// writes traces into files, deletes too old files and monitors hdd usage
{attribute 'reflection'}
FUNCTION_BLOCK PUBLIC FB_TraceHandler IMPLEMENTS I_TraceHandler
(**************************************************************************************
 *  Application     : BoxControl Framework
 *  Revision        : $Revision: 404529 $
 *  Revision date   : $Date: 2020-10-20 08:21:38 +0200 (Mo., 20 Oct 2020) $
 *  Last changed by : $Author: b7lipim $
 *  URL             : $URL: http://almscdc.swisslog.com/repo/SWPD/Development/BoxControlFramework/20_Release/trunk/01_Software/BCF/BCF/JumpStart/20_Product/10_App/11_Com/10_Lib/FB_DebugMsg.TcPOU $
 *
 *  Purpose :	writes (debug) messages into files in subfolders
 *            deletes all subfolders including files older than 7d (according to name, not date)
 *            monitors hdd usage, reports it via debug message and surpress further writing if 80% is exceeded
 *
 * ------------------------------------------------------------------------------------
 *  Copyright Swisslog [IP AG], Switzerland. All rights reserved.
 * 
 * ------------------------------------------------------------------------------------
 *	
 * 	Revision History: 
 *
 *  VERSION DATE         INITIALS     DESCRIPTION
 *  0.0     DD.MM.YYYY   (name)       (explain customized modifications)
 *
 **************************************************************************************)

(********************************************************************************************************************************)
VAR_STAT CONSTANT
  SHELF_LIFE            : TIME                             := T#7D;      // duration until old folders will be deleted
  (*----------------------------------------------------------------------------------------------------------------------------*)
  MAX_FILEOPEN_TIME     : TIME                             := T#100MS;   // maximum file open time until reopen/flush
  LOCKTIME              : TIME                             := T#100MS;   // inhibit time between write attemts
  (*----------------------------------------------------------------------------------------------------------------------------*)
  BUFFER_SIZE           : WORD                             := 8192;      // size of internal file write buffer
  FIFO_SIZE             : WORD                             := 1024;      // size of internal dynamic fifo to temporary store trace entries
  (*----------------------------------------------------------------------------------------------------------------------------*)
  HDD_WARNING_LEVEL     : BYTE                             := 60;        // warning if hdd usage exceeds this percentage
  HDD_ERROR_LEVEL       : BYTE                             := 80;        // error and stop writing if hdd usage exceeds this percentage
END_VAR

(********************************************************************************************************************************)
VAR
  {attribute 'instance-path'}
  {attribute 'no_init'}
  _Instance             : STRING[255]                      := '';         // instance path
  (*----------------------------------------------------------------------------------------------------------------------------*)
  _Enable               : BOOL                             := FALSE;      // HI = writing/deleting enabled
  _MaxFileSizeKB        : WORD                             := 10_240;     // maximum file size in kilobytes
  _Folder               : A_TracePath                      := '';         // working folder without ending '/'
  (*-- duration ----------------------------------------------------------------------------------------------------------------*)
  _StartSystemTick      : ULINT                            := 0;          // system tick at execution start
  _GetSystemTicks       : GETCPUCOUNTER;                                  // Gets the system time in 100ns ticks  
  (*-- general -----------------------------------------------------------------------------------------------------------------*)
  _GetHostName          : FB_GetHostName()                 := (sNetID:= '', tTimeout:= DEFAULT_ADS_TIMEOUT);
  _GetAdaptersInfo      : FB_GetAdaptersInfo()             := (sNetID:= '', tTimeout:= DEFAULT_ADS_TIMEOUT);
  _GetDeviceIdentificationEx : FB_GetDeviceIdentificationEx:= (sNetID:= '', tTimeout:= DEFAULT_ADS_TIMEOUT);
  _MainFolder           : A_TracePath                      := '';         // working folder ending without '/'
  _Active               : BOOL                             := FALSE;      // HI = enable and working folder exists
  _Opened               : BOOL                             := FALSE;      // HI = file is currently open
  _PlcRestarted         : BOOL                             := TRUE;       // HI = add separation lines to file
  _MillisecondsLast		: WORD                             := 16#FFFF;    // system clock monitoring
  _Text                 : STRING[255]                      := '';         // own debug message
  (*-- checking work folder - states -------------------------------------------------------------------------------------------*)
  _CheckState           : E_TraceCheckStates               := E_TraceCheckStates.Initialization;
  _CheckStateLast       : E_TraceCheckStates               := E_TraceCheckStates.Initialization;
  _CheckTime            : TIME                             := T#0S;
  (*-- writing files - states --------------------------------------------------------------------------------------------------*)
  _WriteState           : E_TraceWriteStates               := E_TraceWriteStates.Initialization;
  _WriteStateLast       : E_TraceWriteStates               := E_TraceWriteStates.Initialization;
  _WriteTime            : TIME                             := T#0S;
  (*-- deleting files - states -------------------------------------------------------------------------------------------------*)
  _DeleteState          : E_TraceDeleteStates              := E_TraceDeleteStates.Initialization;
  _DeleteStateLast      : E_TraceDeleteStates              := E_TraceDeleteStates.Initialization;
  _DeleteTime           : TIME                             := T#0S;
  (*-- hdd monitoring ----------------------------------------------------------------------------------------------------------*)
  _HddUsage             : FB_HddUsage;
  _HddUsageTime         : TIME                             := T#0S;
  _HddUsageCount        : DWORD                            := 0;               // counter
  _HddState             : E_TraceHddUsageStates            := E_TraceHddUsageStates.Initialization;
  _HddStateLast         : E_TraceHddUsageStates            := E_TraceHddUsageStates.Initialization;
  _HddTooFull           : BOOL                             := FALSE;           // hdd is too full to write
  _HddFullMissed        : ULINT                            := 0;               // rejected messages due to hdd too full  ( maybe persistent? )
  (*-- writing files - data ----------------------------------------------------------------------------------------------------*)
  _WritePath            : A_TracePath                      := '';              // current working folder with date and trailing '/'
  _WriteFileName        : A_TracePath                      := '';              // current file name
  _WriteDate            : TIMESTRUCT;                                          // current working date
  (*-- file handling -----------------------------------------------------------------------------------------------------------*)
  _FileSize             : ULINT                            := 0;               // current file size in bytes
  _FileIndex            : WORD                             := 0;               // current file number
  _FileTimeOpened       : TIME                             := T#0S;            // timestamp file was opened
  _CreateDir            : Tc2_System.FB_CreateDir;                             // create new folder
  _FileCheck            : Tc2_Utilities.FB_EnumFindFileEntry;                  // checks current working folder for already existing files
  _FileOpen             : Tc2_System.FB_FileOpen;                              // open/create file
  _FileWrite            : Tc2_System.FB_FileWrite;                             // write into file
  _FileClose            : Tc2_System.FB_FileClose;                             // close file
  (*-- folder handling ---------------------------------------------------------------------------------------------------------*)
  _CheckWorkFolder      : Tc2_Utilities.FB_EnumFindFileEntry;                  // checks working folder being existent
  _ScanSubFolder        : Tc2_Utilities.FB_EnumFindFileEntry;                  // checks current working folder for subfolders
  _FileFind             : Tc2_Utilities.FB_EnumFindFileEntry;                  // checks (old) subfolders for files to delete
  _FileDelete           : Tc2_System.FB_FileDelete;                            // delete file
  _FolderRemove         : Tc2_System.FB_RemoveDir;                             // delete folder
  (*-- write fifo --------------------------------------------------------------------------------------------------------------*)
  _TaskCounter          : WORD                             := 0;               // counter for put calls within one plc cycle
  _FifoFillLevel        : WORD                             := 0;               // fill level
  _FifoInput            : WORD                             := 0;               // (next) input position
  _FifoOutput           : WORD                             := 0;               // (next) output position
  _Fifo                 : ARRAY[0..FIFO_SIZE-1] OF POINTER TO FB_TraceEntry;          // fifo itself
  (*-- write data --------------------------------------------------------------------------------------------------------------*)
  _DataDateChanged      : BOOL                             := FALSE;           // date of write data has changed
  _DataLength           : DWORD                            := 0;               // valid length of _DataBuffer
  _DataBuffer           : ARRAY[0..BUFFER_SIZE-1] OF BYTE;                     // data buffer to write into file
  (*-- diagnostics & statisticals ------------------------------------------------------------------------------------------------*)
  _Statistics           : FB_TraceHandlerStatistics();
  _ExecutionDuration    : ULINT                            := 0;               // duration of execution in microseconds
  _ExecutionNow         : ULINT                            := 0;
  (*-- testing -------------------------------------------------------------------------------------------------------------------*)
  _Diag_SystemTime      : ULINT                            := 0;
  _Diag_NoMemory        : ULINT                            := 0;
  _Diag_NoEntry         : ULINT                            := 0;
  _Diag_FifoFull        : ULINT                            := 0;
  _Diag_InvalidDate     : ULINT                            := 0;
END_VAR

(*****************************************************1*********2*********3*********4*********5*********6*********7*********8****)
VAR_STAT CONSTANT                          // 123456789012345678901234567890123456789012345678901234567890123456789012345678900123456789001234567890
{attribute 'hide'}  EOF      : STRING[ 95]:= ';-- end of file ----------------------------------------------------------------';
{attribute 'hide'}  NEWLINE  : STRING[  3]:= '$0D$0A';
{attribute 'hide'}  DIVIDER  : STRING[ 95]:= ';-------------------------------------------------------------------------------';
{attribute 'hide'}  CREATED  : STRING[ 15]:= '; CREATED  : ';
{attribute 'hide'}  TD       : STRING[ 15]:= '; DATE     : ';
{attribute 'hide'}  ENCODING : STRING[ 19]:= '; ENCODING : UTF08';
{attribute 'hide'}  EMPTYLINE: STRING[  3]:= '; ';
{attribute 'hide'}  APPL     : STRING[ 15]:= '; APPL     : ';
{attribute 'hide'}  BUILD    : STRING[ 15]:= '; BUILD    : ';
{attribute 'hide'}  HOST     : STRING[ 15]:= '; HOST     : ';
{attribute 'hide'}  ADDR     : STRING[ 15]:= '; ADDR     : ';
{attribute 'hide'}  OPSYSTEM : STRING[ 15]:= '; SYSTEM   : ';
{attribute 'hide'}  RUNTIME  : STRING[ 19]:= '; RUNTIME  : TC';
{attribute 'hide'}  INFO     : STRING[ 15]:= '; INFO     : ';
{attribute 'hide'}  SIZE     : STRING[ 15]:= '; SIZE     : ';
{attribute 'hide'}  HEADER   : STRING[195]:= '; -- DATE & TIME ------- count -- level -- instance -------------------------- position ------- message ------- additional information ------';
END_VAR


(********************************************************************************************************************************)
(** calculate execution time ****************************************************************************************************)
_GetSystemTicks();
_StartSystemTick:= (         DWORD_TO_ULINT(_GetSystemTicks.cpuCntLoDW)
                     OR SHL( DWORD_TO_ULINT(_GetSystemTicks.cpuCntHiDW),  32 )  );




(********************************************************************************************************************************)
(** run all services ************************************************************************************************************)
_HddUsage();  // call here to use everywhere

M_RunHddUsage();
M_RunCheck();
M_RunWrite();
M_RunDelete();

IF (_MillisecondsLast = System.fbSystemTime.TIMESTR.wMilliseconds)
THEN
  _Diag_SystemTime:= _Diag_SystemTime + 1;

  (*-- trace it ---------------------------------------------------*)
  IF(_TaskCounter <> 0)
  THEN
// example: '11-000-0000-00-0,  system time not updated'
   ;(* _Text:= '';
    _Text:= CONCAT(_Text, F_AddDividerToSisString(SubsystemRegistry.SubsystemName) );
    _Text:= CONCAT(_Text, ',  system time not updated');
    Put( MsgType := E_DebugMsgType.WARNING,
         Instance:= ADR(_Instance),
         Text    := ADR(_Text)  );*)
  END_IF
END_IF

_MillisecondsLast:= System.fbSystemTime.TIMESTR.wMilliseconds;
_TaskCounter:= 0;




(********************************************************************************************************************************)
(** calculate execution time ****************************************************************************************************)
_GetSystemTicks();

_ExecutionNow:= (         DWORD_TO_ULINT(_GetSystemTicks.cpuCntLoDW)
                  OR SHL( DWORD_TO_ULINT(_GetSystemTicks.cpuCntHiDW),  32 )  );

_ExecutionDuration:= (_ExecutionNow - _StartSystemTick + 5) / 10;

_Statistics.MaxExecutionDuration:= MAX(_Statistics.MaxExecutionDuration, _ExecutionDuration);




(********************************************************************************************************************************)
(** done ************************************************************************************************************************)

// clears the internal fifo (all unwritten traces will be lost)
METHOD PUBLIC Clear

(********************************************************************************************************************************)
VAR_INPUT
END_VAR

(********************************************************************************************************************************)
VAR
  Index                 : WORD                             := 0;
  Entry                 : POINTER TO FB_TraceEntry         := 0;
END_VAR

(********************************************************************************************************************************)
(********************************************************************************************************************************)
_FifoFillLevel:= 0;
_FifoInput    := 0;
_FifoOutput   := 0;




(********************************************************************************************************************************)
(********************************************************************************************************************************)
Index:= 0;
WHILE (Index < FIFO_SIZE)
DO
  Entry:= _Fifo[Index];

  (*-- release memory -----------------------------------------------*)
  IF (Entry <> 0)
  THEN
    __DELETE(Entry);
  END_IF

  (*-- next ---------------------------------------------------------*)
  _Fifo[Index]:= 0;
  Index:= Index + 1;
END_WHILE




(********************************************************************************************************************************)
(** done ************************************************************************************************************************)
END_METHOD

// HI = writing/deleting enabled
{attribute 'monitoring' := 'call'}
PROPERTY PUBLIC Enable : BOOL
GET
Enable:= _Enable;
END_GET
SET
(********************************************************************************************************************************)
(** change? *********************************************************************************************************************)
IF (_Enable = Enable)
THEN
  RETURN;
END_IF

_Enable:= Enable;




(********************************************************************************************************************************)
(** done ************************************************************************************************************************)
END_SET
END_PROPERTY

{attribute 'hide'}
METHOD FB_exit : BOOL

(********************************************************************************************************************************)
VAR_INPUT
	bInCopyCode           : BOOL;  // if TRUE, the instance afterwards gets moved into the copy code (online change)
  (*----------------------------------------------------------------------------------------------------------------------------*)
END_VAR

(********************************************************************************************************************************)
(** release dynamically assigned memory *****************************************************************************************)
Clear();




(********************************************************************************************************************************)
(** done ************************************************************************************************************************)
END_METHOD

{attribute 'hide'}
METHOD FB_init : BOOL

(********************************************************************************************************************************)
VAR_INPUT
	bInitRetains          : BOOL; // if TRUE, the retain variables are initialized (warm start / cold start)
	bInCopyCode           : BOOL;  // if TRUE, the instance afterwards gets moved into the copy code (online change)
  (*----------------------------------------------------------------------------------------------------------------------------*)
END_VAR

(********************************************************************************************************************************)
VAR
END_VAR

(********************************************************************************************************************************)
(** remove 'QB2Jumpstart.JumpStart.' from instance path *************************************************************************)
F_InstancePathRemovals( DestStart     := ADR(_Instance),
                        DestEnd       := ADR(_Instance) + SIZEOF(_Instance),
                        RemoveLastPart:= FALSE );




(********************************************************************************************************************************)
(** done ************************************************************************************************************************)
END_METHOD

// folder to work within, folder must exist! (will only take effect when enabled is low)
{attribute 'monitoring' := 'call'}
PROPERTY PUBLIC Folder : A_TracePath
GET
Folder:= _Folder;
END_GET
SET
VAR
  Idx                   : WORD                             := 0;
  SepFound              : BOOL                             := FALSE;
  Finished              : BOOL                             := FALSE;
END_VAR
(********************************************************************************************************************************)
(** change? *********************************************************************************************************************)
IF (_Folder = Folder)
THEN
  RETURN;
END_IF

_Folder:= Folder;




(********************************************************************************************************************************)
(** change '\' to '/' and remove a trailing '/' if neccessary *******************************************************************)
Idx:= 0;
WHILE (Idx < SIZEOF(_Folder)  )
DO
  (*-- replace '\' with '/' -------------------------------------------------------------*)
  IF (_Folder[Idx] = 16#5C)  (* '\' *)
  THEN
    _Folder[Idx]:= 16#2F;   (* '/' *)
    SepFound:= TRUE;

  (*-- separation found '/' -------------------------------------------------------------*)
  ELSIF(_Folder[Idx] = 16#2F)   (* '/' *)
  THEN
    SepFound:= TRUE;

  (*-- fill rest of string with terminations --------------------------------------------*)
  ELSIF(Finished = TRUE)
  THEN
    (*-------------------------------------------*)
    _Folder[Idx]:= 16#00;

  (*-- string termination found ---------------------------------------------------------*)
  ELSIF(_Folder[Idx] = 16#00)
  THEN
    (*-- remove trailing '/' --------------------*)
    IF (SepFound = TRUE)
    THEN
      _Folder[Idx-1] := 16#00;
    END_IF
    (*-------------------------------------------*)
    Finished:= TRUE;
    SepFound:= FALSE;

  (*-- normal character -----------------------------------------------------------------*)
  ELSE
    SepFound:= FALSE;
  END_IF

  (*-- next -----------------------------------------------------------------------------*)
  Idx:= Idx + 1;
END_WHILE




(********************************************************************************************************************************)
(** done ************************************************************************************************************************)
END_SET
END_PROPERTY

// usage/free and total space of hdd
{attribute 'monitoring' := 'call'}
PROPERTY PUBLIC HddUsage : I_HddUsage
GET
HddUsage:= _HddUsage;
END_GET
END_PROPERTY

// builds the file name with index
METHOD PROTECTED M_BuildFileName

(********************************************************************************************************************************)
VAR
  DestStart             : POINTER TO BYTE                  := 0;     // start position to concat
  DestEnd               : POINTER TO BYTE                  := 0;     // buffer/string end
END_VAR

(********************************************************************************************************************************)
(********************************************************************************************************************************)
DestStart:= ADR(_WriteFileName);
DestEnd  := ADR(_WriteFileName) + SIZEOF(_WriteFileName);

(*-- application ---------------------------------------------------------------------------------------------------------------*)
DestStart:= F_StringCopy          ( DestStart:= DestStart,  DestEnd:= DestEnd,  Source    := ADR(_GetHostName.sHostName)  );

(*-- date ----------------------------------------------------------------------------------------------------------------------*)
DestStart:= F_StringCopy          ( DestStart:= DestStart,  DestEnd:= DestEnd,  Source    := ADR('_')  );
DestStart:= F_StringFromDatestruct( DestStart:= DestStart,  DestEnd:= DestEnd,  DateStruct:= _WriteDate );

(*-- index ---------------------------------------------------------------------------------------------------------------------*)
DestStart:= F_StringCopy          ( DestStart:= DestStart,  DestEnd:= DestEnd,  Source    := ADR('_')  );
DestStart:= F_StringFromWord      ( DestStart:= DestStart,  DestEnd:= DestEnd,  Value     := _FileIndex,  Length:= 4 );


(*-- file type -----------------------------------------------------------------------------------------------------------------*)
DestStart:= F_StringCopy          ( DestStart:= DestStart,  DestEnd:= DestEnd,  Source    := ADR('_Trace.txt')  );




(********************************************************************************************************************************)
(** done ************************************************************************************************************************)
END_METHOD

// created data to write, returns TRUE if trace date has changed
METHOD PROTECTED M_CreateData : BOOL

(********************************************************************************************************************************)
VAR
  MsgText               : STRING[31]                       := ''; 
  (*----------------------------------------------------------------------------------------------------------------------------*)
  DestStart             : POINTER TO BYTE                  := 0;
  DestWork              : POINTER TO BYTE                  := 0;
  DestEnd               : POINTER TO BYTE                  := 0;
  (*----------------------------------------------------------------------------------------------------------------------------*)
  EntryStart            : POINTER TO BYTE                  := 0;
  Entry                 : POINTER TO FB_TraceEntry         := 0;
  DateChanged           : BOOL                             := FALSE;
  Count                 : WORD                             := 0;
END_VAR

(********************************************************************************************************************************)
(********************************************************************************************************************************)
_DataLength:= 0;

DestStart:= ADR(_DataBuffer);
DestWork := ADR(_DataBuffer);
DestEnd  := ADR(_DataBuffer) + SIZEOF(_DataBuffer);

DateChanged:= FALSE;




(********************************************************************************************************************************)
(********************************************************************************************************************************)
Count:= 0;
WHILE(_FifoFillLevel <> 0)
DO
  (*-- get new entry --------------------------------------------------------------------*)
  Entry:= _Fifo[_FifoOutput];
  IF (Entry = 0)
  THEN
    EXIT;
  END_IF

  (*-- entry has already new date? ------------------------------------------------------*)
  IF (Entry^.IsEqualDate(_WriteDate) = FALSE)
  THEN
    DateChanged:= TRUE;
    EXIT;
  END_IF

  (*-- prepare line ---------------------------------------------------------------------*)
  MsgText:= TO_STRING(Entry^.MsgType);

  (*-- build line -----------------------------------------------------------------------*)
  EntryStart:= DestWork;
  DestWork:= F_StringFromDatestruct( DestStart:= DestWork,  DestEnd:= DestEnd,  DateStruct:= Entry^.DateTime  );
  DestWork:= F_StringCopy          ( DestStart:= DestWork,  DestEnd:= DestEnd,  Source    := ADR('  ')  );
  DestWork:= F_StringFromTimestruct( DestStart:= DestWork,  DestEnd:= DestEnd,  TimeStruct:= Entry^.DateTime,     ShowMs:= TRUE  );
  DestWork:= F_StringCopy          ( DestStart:= DestWork,  DestEnd:= DestEnd,  Source    := ADR(':  ')  );
  DestWork:= F_StringFromWord      ( DestStart:= DestWork,  DestEnd:= DestEnd,  Value     := Entry^.TaskCounter,  Length:= 0  );
  DestWork:= F_StringCopy          ( DestStart:= DestWork,  DestEnd:= DestEnd,  Source    := ADR(' = ')  );
  DestWork:= F_StringCopy          ( DestStart:= DestWork,  DestEnd:= DestEnd,  Source    := ADR(MsgText)  );
  DestWork:= F_StringCopy          ( DestStart:= DestWork,  DestEnd:= DestEnd,  Source    := ADR(',  ')  );
  DestWork:= F_StringCopy          ( DestStart:= DestWork,  DestEnd:= DestEnd,  Source    := Entry^.InstancePtr); 
  DestWork:= F_StringCopy          ( DestStart:= DestWork,  DestEnd:= DestEnd,  Source    := ADR(',  ')  );
  DestWork:= F_StringCopy          ( DestStart:= DestWork,  DestEnd:= DestEnd,  Source    := Entry^.TextPtr ); 
  DestWork:= F_StringCopy          ( DestStart:= DestWork,  DestEnd:= DestEnd,  Source    := ADR(NEWLINE)  );

  (*-- did not fit into write buffer (anymore) ------------------------------------------*)
  IF (DestWork >= DestEnd - 1)
  THEN
    DestWork:= EntryStart;
    EXIT;
  END_IF

  (*-- remove from fifo -----------------------------------------------------------------*)
  __DELETE(Entry);
  _Fifo[_FifoOutput]:= 0;

  (*-- next entry -> actualize fifo -----------------------------------------------------*)
  _FifoOutput:= _FifoOutput + 1;
  IF (_FifoOutput    >= FIFO_SIZE)  THEN  _FifoOutput:= 0;  END_IF
  IF (_FifoFillLevel > 0)           THEN  _FifoFillLevel:= _FifoFillLevel - 1;  END_IF

  (*-------------------------------------------------------------------------------------*)
  Count:= Count + 1;
END_WHILE

_Statistics.MaxDataItemsPerRow:= MAX(_Statistics.MaxDataItemsPerRow, Count);




(********************************************************************************************************************************)
(** calculate data length *******************************************************************************************************)
_DataLength:= (DestWork - DestStart);

_Statistics.MaxDataLength:= MAX(_Statistics.MaxDataLength, _DataLength);




(********************************************************************************************************************************)
(** done ************************************************************************************************************************)
M_CreateData:= DateChanged;
END_METHOD

// creates the eof file end
METHOD PROTECTED M_CreateEof

(********************************************************************************************************************************)
VAR
  DestStart             : POINTER TO BYTE                  := 0;
  DestWork              : POINTER TO BYTE                  := 0;
  DestEnd               : POINTER TO BYTE                  := 0;
END_VAR

(********************************************************************************************************************************)
(********************************************************************************************************************************)
_DataLength:= 0;

DestStart:= ADR(_DataBuffer);
DestWork := ADR(_DataBuffer);
DestEnd  := ADR(_DataBuffer) + SIZEOF(_DataBuffer);




(********************************************************************************************************************************)
(********************************************************************************************************************************)
DestWork:= F_StringCopy(DestStart:= DestWork, DestEnd:= DestEnd, Source:= ADR(NEWLINE)  );
DestWork:= F_StringCopy(DestStart:= DestWork, DestEnd:= DestEnd, Source:= ADR(EOF)      );
DestWork:= F_StringCopy(DestStart:= DestWork, DestEnd:= DestEnd, Source:= ADR(NEWLINE)  );
DestWork:= F_StringCopy(DestStart:= DestWork, DestEnd:= DestEnd, Source:= ADR(NEWLINE)  );




(********************************************************************************************************************************)
(** calculate data length *******************************************************************************************************)
_DataLength:= (DestWork - DestStart);

_Statistics.MaxDataLength:= MAX(_Statistics.MaxDataLength, _DataLength);




(********************************************************************************************************************************)
(** done ************************************************************************************************************************)
END_METHOD

// creates the file header for a new file
METHOD PROTECTED M_CreateHeader

(********************************************************************************************************************************)
VAR
  DestStart             : POINTER TO BYTE                  := 0;
  DestWork              : POINTER TO BYTE                  := 0;
  DestEnd               : POINTER TO BYTE                  := 0;
  (*----------------------------------------------------------------------------------------------------------------------------*)
  AdapterInfo           : ST_IpAdapterInfo;
  Idx                   : BYTE                             := 0;
END_VAR

(********************************************************************************************************************************)
(********************************************************************************************************************************)
_DataLength:= 0;

DestStart:= ADR(_DataBuffer);
DestWork := ADR(_DataBuffer);
DestEnd  := ADR(_DataBuffer) + SIZEOF(_DataBuffer);




(********************************************************************************************************************************)
(********************************************************************************************************************************)
(*-- ;-line --------------------------------------------------------------------------------------------------------------------*)
DestWork:= F_StringCopy( DestStart:= DestWork,  DestEnd:= DestEnd,  Source:= ADR(DIVIDER)  );
DestWork:= F_StringCopy( DestStart:= DestWork,  DestEnd:= DestEnd,  Source:= ADR(NEWLINE)  );


(*-- info line -----------------------------------------------------------------------------------------------------------------*)
DestWork:= F_StringCopy( DestStart:= DestWork,  DestEnd:= DestEnd,  Source:= ADR(CREATED)            );
DestWork:= F_StringCopy( DestStart:= DestWork,  DestEnd:= DestEnd,  Source:= ADR('FB_TraceHandler')  );
DestWork:= F_StringCopy( DestStart:= DestWork,  DestEnd:= DestEnd,  Source:= ADR('  ')               );
DestWork:= F_StringCopy( DestStart:= DestWork,  DestEnd:= DestEnd,  Source:= ADR('[b7lipim]')        );
DestWork:= F_StringCopy( DestStart:= DestWork,  DestEnd:= DestEnd,  Source:= ADR(NEWLINE)            );


(*-- Datum&Uhrzeit-Zeile bauen -------------------------------------------------------------------------------------------------*)
DestWork:= F_StringCopy          ( DestStart:= DestWork,  DestEnd:= DestEnd,  Source    := ADR(TD)          );
DestWork:= F_StringFromDatestruct( DestStart:= DestWork,  DestEnd:= DestEnd,  DateStruct:= System.fbSystemTime.TIMESTR  );
DestWork:= F_StringCopy          ( DestStart:= DestWork,  DestEnd:= DestEnd,  Source    := ADR('  ')        );
DestWork:= F_StringFromTimestruct( DestStart:= DestWork,  DestEnd:= DestEnd,  TimeStruct:= System.fbSystemTime.TIMESTR, ShowMs:= TRUE  );
DestWork:= F_StringCopy          ( DestStart:= DestWork,  DestEnd:= DestEnd,  Source    := ADR(NEWLINE)     );


(*-- Encoding Info -------------------------------------------------------------------------------------------------------------*)
DestWork:= F_StringCopy( DestStart:= DestWork,  DestEnd:= DestEnd,  Source:= ADR(ENCODING)  );
DestWork:= F_StringCopy( DestStart:= DestWork,  DestEnd:= DestEnd,  Source:= ADR(NEWLINE)   );


(*-- Applikation ---------------------------------------------------------------------------------------------------------------*)
DestWork:= F_StringCopy( DestStart:= DestWork,  DestEnd:= DestEnd,  Source:= ADR(EMPTYLINE) );
DestWork:= F_StringCopy( DestStart:= DestWork,  DestEnd:= DestEnd,  Source:= ADR(NEWLINE)   );
DestWork:= F_StringCopy( DestStart:= DestWork,  DestEnd:= DestEnd,  Source:= ADR(APPL)      );
DestWork:= F_StringCopy( DestStart:= DestWork,  DestEnd:= DestEnd,  Source:= ADR('??')      );
DestWork:= F_StringCopy( DestStart:= DestWork,  DestEnd:= DestEnd,  Source:= ADR('  ')      );
DestWork:= F_StringCopy( DestStart:= DestWork,  DestEnd:= DestEnd,  Source:= ADR('??')      );
DestWork:= F_StringCopy( DestStart:= DestWork,  DestEnd:= DestEnd,  Source:= ADR('  (')     );
DestWork:= F_StringCopy( DestStart:= DestWork,  DestEnd:= DestEnd,  Source:= ADR('??')      );
DestWork:= F_StringCopy( DestStart:= DestWork,  DestEnd:= DestEnd,  Source:= ADR(')' )      );
DestWork:= F_StringCopy( DestStart:= DestWork,  DestEnd:= DestEnd,  Source:= ADR(NEWLINE)   );


(*-- Build ---------------------------------------------------------------------------------------------------------------------*)


(*-- Host/Addr -----------------------------------------------------------------------------------------------------------------*)
DestWork:= F_StringCopy( DestStart:= DestWork,  DestEnd:= DestEnd,  Source:= ADR(EMPTYLINE) );
DestWork:= F_StringCopy( DestStart:= DestWork,  DestEnd:= DestEnd,  Source:= ADR(NEWLINE)   );
DestWork:= F_StringCopy( DestStart:= DestWork,  DestEnd:= DestEnd,  Source:= ADR(HOST)      );
DestWork:= F_StringCopy( DestStart:= DestWork,  DestEnd:= DestEnd,  Source:= ADR(_GetHostName.sHostName)  );
DestWork:= F_StringCopy( DestStart:= DestWork,  DestEnd:= DestEnd,  Source:= ADR(' @')      );
DestWork:= F_StringCopy( DestStart:= DestWork,  DestEnd:= DestEnd,  Source:= ADR(_GetDeviceIdentificationEx.stDevIdent.strAmsNetId) );
DestWork:= F_StringCopy( DestStart:= DestWork,  DestEnd:= DestEnd,  Source:= ADR(NEWLINE)   );

Idx:= 0;
WHILE(Idx <= Tc2_Utilities.MAX_LOCAL_ADAPTERS)
DO
  AdapterInfo:= _GetAdaptersInfo.arrAdapters[Idx];
  Idx:= Idx + 1;
  (*-- valid? ---------------------------------------------------------------------------*)
  IF(AdapterInfo.sIpAddr = '')         THEN  CONTINUE;  END_IF
  IF(AdapterInfo.sIpAddr = '0.0.0.0')  THEN  CONTINUE;  END_IF
  (*-------------------------------------------------------------------------------------*)
  DestWork:= F_StringCopy( DestStart:= DestWork,  DestEnd:= DestEnd,  Source:= ADR(ADDR)      );
  DestWork:= F_StringCopy( DestStart:= DestWork,  DestEnd:= DestEnd,  Source:= ADR(AdapterInfo.sIpAddr) );
  DestWork:= F_StringCopy( DestStart:= DestWork,  DestEnd:= DestEnd,  Source:= ADR('/') );
  DestWork:= F_StringCopy( DestStart:= DestWork,  DestEnd:= DestEnd,  Source:= ADR(AdapterInfo.sSubNet) );
  DestWork:= F_StringCopy( DestStart:= DestWork,  DestEnd:= DestEnd,  Source:= ADR('  {') );
  DestWork:= F_StringCopy( DestStart:= DestWork,  DestEnd:= DestEnd,  Source:= ADR(AdapterInfo.sDescription) );
  DestWork:= F_StringCopy( DestStart:= DestWork,  DestEnd:= DestEnd,  Source:= ADR('}') );
  (*-------------------------------------------------------------------------------------*)
  DestWork:= F_StringCopy( DestStart:= DestWork,  DestEnd:= DestEnd,  Source:= ADR(NEWLINE)   );
END_WHILE


(*-- System --------------------------------------------------------------------------------------------------------------------*)
DestWork:= F_StringCopy( DestStart:= DestWork,  DestEnd:= DestEnd,  Source:= ADR(EMPTYLINE) );
DestWork:= F_StringCopy( DestStart:= DestWork,  DestEnd:= DestEnd,  Source:= ADR(NEWLINE)   );
DestWork:= F_StringCopy( DestStart:= DestWork,  DestEnd:= DestEnd,  Source:= ADR(OPSYSTEM)  );
DestWork:= F_StringCopy( DestStart:= DestWork,  DestEnd:= DestEnd,  Source:= ADR(_GetDeviceIdentificationEx.stDevIdent.strImageOsName)    );
DestWork:= F_StringCopy( DestStart:= DestWork,  DestEnd:= DestEnd,  Source:= ADR('  {')    );
DestWork:= F_StringCopy( DestStart:= DestWork,  DestEnd:= DestEnd,  Source:= ADR(_GetDeviceIdentificationEx.stDevIdent.strImageOsVersion)    );
DestWork:= F_StringCopy( DestStart:= DestWork,  DestEnd:= DestEnd,  Source:= ADR('}')    );
DestWork:= F_StringCopy( DestStart:= DestWork,  DestEnd:= DestEnd,  Source:= ADR(NEWLINE)   );
DestWork:= F_StringCopy( DestStart:= DestWork,  DestEnd:= DestEnd,  Source:= ADR(RUNTIME)   );
DestWork:= F_StringCopy( DestStart:= DestWork,  DestEnd:= DestEnd,  Source:= ADR(_GetDeviceIdentificationEx.stDevIdent.strTwinCATVersion)    );
DestWork:= F_StringCopy( DestStart:= DestWork,  DestEnd:= DestEnd,  Source:= ADR('.')    );
DestWork:= F_StringCopy( DestStart:= DestWork,  DestEnd:= DestEnd,  Source:= ADR(_GetDeviceIdentificationEx.stDevIdent.strTwinCATRevision)   );
DestWork:= F_StringCopy( DestStart:= DestWork,  DestEnd:= DestEnd,  Source:= ADR('.')    );
DestWork:= F_StringCopy( DestStart:= DestWork,  DestEnd:= DestEnd,  Source:= ADR(_GetDeviceIdentificationEx.stDevIdent.strTwinCATBuild)      );
DestWork:= F_StringCopy( DestStart:= DestWork,  DestEnd:= DestEnd,  Source:= ADR(NEWLINE)         );



(*-- Info ----------------------------------------------------------------------------------------------------------------------*)
DestWork:= F_StringCopy    ( DestStart:= DestWork,  DestEnd:= DestEnd,  Source:= ADR(EMPTYLINE)       );
DestWork:= F_StringCopy    ( DestStart:= DestWork,  DestEnd:= DestEnd,  Source:= ADR(NEWLINE)         );
DestWork:= F_StringCopy    ( DestStart:= DestWork,  DestEnd:= DestEnd,  Source:= ADR(INFO)            );
DestWork:= F_StringCopy    ( DestStart:= DestWork,  DestEnd:= DestEnd,  Source:= ADR(_WriteFileName)  );
DestWork:= F_StringCopy    ( DestStart:= DestWork,  DestEnd:= DestEnd,  Source:= ADR(NEWLINE)         );
DestWork:= F_StringCopy    ( DestStart:= DestWork,  DestEnd:= DestEnd,  Source:= ADR(SIZE)            );
DestWork:= F_StringCopy    ( DestStart:= DestWork,  DestEnd:= DestEnd,  Source:= ADR('<= ')           );
DestWork:= F_StringFromWord( DestStart:= DestWork,  DestEnd:= DestEnd,  Value := _MaxFileSizeKB,  Length:= 0  );
DestWork:= F_StringCopy    ( DestStart:= DestWork,  DestEnd:= DestEnd,  Source:= ADR('kB')            );
DestWork:= F_StringCopy    ( DestStart:= DestWork,  DestEnd:= DestEnd,  Source:= ADR(NEWLINE)         );


(*-- ;-line --------------------------------------------------------------------------------------------------------------------*)
DestWork:= F_StringCopy( DestStart:= DestWork,  DestEnd:= DestEnd,  Source:= ADR(DIVIDER)  );
DestWork:= F_StringCopy( DestStart:= DestWork,  DestEnd:= DestEnd,  Source:= ADR(NEWLINE)  );




(********************************************************************************************************************************)
(** table header ****************************************************************************************************************)
DestWork:= F_StringCopy( DestStart:= DestWork,  DestEnd:= DestEnd,  Source:= ADR(NEWLINE)  );
DestWork:= F_StringCopy( DestStart:= DestWork,  DestEnd:= DestEnd,  Source:= ADR(NEWLINE)  );
DestWork:= F_StringCopy( DestStart:= DestWork,  DestEnd:= DestEnd,  Source:= ADR(HEADER)   );
DestWork:= F_StringCopy( DestStart:= DestWork,  DestEnd:= DestEnd,  Source:= ADR(NEWLINE)  );
DestWork:= F_StringCopy( DestStart:= DestWork,  DestEnd:= DestEnd,  Source:= ADR(NEWLINE)  );




(********************************************************************************************************************************)
(** calculate data length *******************************************************************************************************)
_DataLength:= (DestWork - DestStart);

_Statistics.MaxDataLength:= MAX(_Statistics.MaxDataLength, _DataLength);




(********************************************************************************************************************************)
(** done ************************************************************************************************************************)
END_METHOD

METHOD PROTECTED M_CreatePlcDivider

(********************************************************************************************************************************)
VAR
  DestStart             : POINTER TO BYTE                  := 0;
  DestWork              : POINTER TO BYTE                  := 0;
  DestEnd               : POINTER TO BYTE                  := 0;
  (*----------------------------------------------------------------------------------------------------------------------------*)
  DateString            : STRING[15]                       := '';
  TimeString            : STRING[15]                       := '';
  FileSize              : STRING[15]                       := '';
END_VAR

(********************************************************************************************************************************)
(********************************************************************************************************************************)
_DataLength:= 0;

DestStart:= ADR(_DataBuffer);
DestWork := ADR(_DataBuffer);
DestEnd  := ADR(_DataBuffer) + SIZEOF(_DataBuffer);




(********************************************************************************************************************************)
(********************************************************************************************************************************)
DestWork:= F_StringCopy(DestStart:= DestWork, DestEnd:= DestEnd, Source:= ADR(NEWLINE)  );
DestWork:= F_StringCopy(DestStart:= DestWork, DestEnd:= DestEnd, Source:= ADR(NEWLINE)  );




(********************************************************************************************************************************)
(** calculate data length *******************************************************************************************************)
_DataLength:= (DestWork - DestStart);

_Statistics.MaxDataLength:= MAX(_Statistics.MaxDataLength, _DataLength);




(********************************************************************************************************************************)
(** done ************************************************************************************************************************)
END_METHOD

// checks existence of working folder
METHOD PROTECTED M_RunCheck

(********************************************************************************************************************************)
VAR
END_VAR

(********************************************************************************************************************************)
(** initialization **************************************************************************************************************)
CASE(_CheckState) OF
E_TraceCheckStates.Initialization:
  (*-- ENTRY -------------------------------------------------------------------------------------------------------------------*)
    _CheckStateLast:= _CheckState;

  (*-- ACTION ------------------------------------------------------------------------------------------------------------------*)

  (*-- TRANSITION --------------------------------------------------------------------------------------------------------------*)
  _CheckState:= E_TraceCheckStates.Delay;




(********************************************************************************************************************************)
(** short delay *****************************************************************************************************************)
E_TraceCheckStates.Delay:
  (*-- ENTRY -------------------------------------------------------------------------------------------------------------------*)
  IF (_CheckStateLast <> _CheckState)
  THEN
    _CheckStateLast:= _CheckState;
    _CheckTime     := F_GetTimeMsTick();
    (*-----------------------------------------------------------------------------------*)
  END_IF

  (*-- ACTION ------------------------------------------------------------------------------------------------------------------*)

  (*-- TRANSITION --------------------------------------------------------------------------------------------------------------*)
  (*-- delay time over ------------------------------------------------------------------*)
  IF(F_GetTimeMsDiff(_CheckTime) >= T#1S)
  THEN
    _CheckState:= E_TraceCheckStates.Hostname;
  END_IF




(********************************************************************************************************************************)
(** retrieve hostname ***********************************************************************************************************)
E_TraceCheckStates.Hostname:
  (*-- ENTRY -------------------------------------------------------------------------------------------------------------------*)
  IF (_CheckStateLast <> _CheckState)
  THEN
    _CheckStateLast:= _CheckState;
    _CheckTime     := F_GetTimeMsTick();
    (*-----------------------------------------------------------------------------------*)
    _GetHostName(bExecute:= FALSE);
    _GetHostName.bExecute:= TRUE;
  END_IF

  (*-- ACTION ------------------------------------------------------------------------------------------------------------------*)
  _GetHostName();

  (*-- TRANSITION --------------------------------------------------------------------------------------------------------------*)
  IF (_GetHostName.bBusy = FALSE)
  THEN
    _CheckState:= E_TraceCheckStates.Adapters;
  END_IF




(********************************************************************************************************************************)
(** retrieve network adapters infos *********************************************************************************************)
E_TraceCheckStates.Adapters:
  (*-- ENTRY -------------------------------------------------------------------------------------------------------------------*)
  IF (_CheckStateLast <> _CheckState)
  THEN
    _CheckStateLast:= _CheckState;
    _CheckTime     := F_GetTimeMsTick();
    (*-----------------------------------------------------------------------------------*)
    _GetAdaptersInfo(bExecute:= FALSE);
    _GetAdaptersInfo.bExecute:= TRUE;
  END_IF

  (*-- ACTION ------------------------------------------------------------------------------------------------------------------*)
  _GetAdaptersInfo();

  (*-- TRANSITION --------------------------------------------------------------------------------------------------------------*)
  IF (_GetAdaptersInfo.bBusy = FALSE)
  THEN
    _CheckState:= E_TraceCheckStates.DeviceIdentification;
  END_IF




(********************************************************************************************************************************)
(** retrieve device identification **********************************************************************************************)
E_TraceCheckStates.DeviceIdentification:
  (*-- ENTRY -------------------------------------------------------------------------------------------------------------------*)
  IF (_CheckStateLast <> _CheckState)
  THEN
    _CheckStateLast:= _CheckState;
    _CheckTime     := F_GetTimeMsTick();
    (*-----------------------------------------------------------------------------------*)
    _GetDeviceIdentificationEx(bExecute:= FALSE);
    _GetDeviceIdentificationEx.bExecute:= TRUE;
  END_IF

  (*-- ACTION ------------------------------------------------------------------------------------------------------------------*)
  _GetDeviceIdentificationEx();

  (*-- TRANSITION --------------------------------------------------------------------------------------------------------------*)
  IF (_GetDeviceIdentificationEx.bBusy = FALSE)
  THEN
    _CheckState:= E_TraceCheckStates.Disabled;
  END_IF




(********************************************************************************************************************************)
(** fb disabled *****************************************************************************************************************)
E_TraceCheckStates.Disabled:
  (*-- ENTRY -------------------------------------------------------------------------------------------------------------------*)
  IF (_CheckStateLast <> _CheckState)
  THEN
    _CheckStateLast:= _CheckState;
    _CheckTime     := F_GetTimeMsTick();
    (*-----------------------------------------------------------------------------------*)
    _Active    := FALSE;
    _MainFolder:= '';
  END_IF

  (*-- ACTION ------------------------------------------------------------------------------------------------------------------*)

  (*-- TRANSITION --------------------------------------------------------------------------------------------------------------*)
  (*-- enabled --------------------------------------------------------------------------*)
  IF (_Enable = TRUE)
  THEN
    _MainFolder:= _Folder;
    (*-------------------------------------------*)
    _CheckState:= E_TraceCheckStates.HddCheck;
  END_IF




(********************************************************************************************************************************)
(** hdd usage read ******************************************************************************************************************************)
E_TraceCheckStates.HddCheck:
  (*-- ENTRY -------------------------------------------------------------------------------------------------------------------*)
  IF (_CheckStateLast <> _CheckState)
  THEN
    _CheckStateLast:= _CheckState;
    _CheckTime     := F_GetTimeMsTick();
    (*-----------------------------------------------------------------------------------*)
  END_IF

  (*-- ACTION ------------------------------------------------------------------------------------------------------------------*)

  (*-- TRANSITION --------------------------------------------------------------------------------------------------------------*)
  IF (F_GetTimeMsDiff(_HddUsageTime) >= T#5M)  THEN  _CheckState:= E_TraceCheckStates.HddUsage;
  ELSE                                               _CheckState:= E_TraceCheckStates.Start;
  END_IF




(********************************************************************************************************************************)
(** read hdd usage **************************************************************************************************************)
E_TraceCheckStates.HddUsage:
  (*-- ENTRY -------------------------------------------------------------------------------------------------------------------*)
  IF (_CheckStateLast <> _CheckState)
  THEN
    _CheckStateLast:= _CheckState;
    _CheckTime     := F_GetTimeMsTick();
    (*-----------------------------------------------------------------------------------*)
    _HddUsage.Start( Drive:= _MainFolder );  // use drive letter from main folder
    _HddUsageTime:= F_GetTimeMsTick();
  END_IF

  (*-- ACTION ------------------------------------------------------------------------------------------------------------------*)
    // _HddUsage() is called in main body to be used in other state machines as well

  (*-- TRANSITION --------------------------------------------------------------------------------------------------------------*)
  IF (_HddUsage.Busy = FALSE)
  THEN
    _HddUsageCount:= _HddUsageCount + 1;
    (*-------------------------------------------*)
    IF    (_HddUsage.Error           = TRUE)               THEN  _HddState:= E_TraceHddUsageStates.Unknown;
    ELSIF (_HddUsage.PercentageUsed >= HDD_ERROR_LEVEL)    THEN  _HddState:= E_TraceHddUsageStates.ErrorLevel;
    ELSIF (_HddUsage.PercentageUsed >= HDD_WARNING_LEVEL)  THEN  _HddState:= E_TraceHddUsageStates.WarningLevel;
    ELSE                                                         _HddState:= E_TraceHddUsageStates.EnoughFree;
    END_IF
    (*-------------------------------------------*)
    _CheckState:= E_TraceCheckStates.Start;
  END_IF




(********************************************************************************************************************************)
(** prepare work folder check ***************************************************************************************************)
E_TraceCheckStates.Start:
  (*-- ENTRY -------------------------------------------------------------------------------------------------------------------*)
  IF (_CheckStateLast <> _CheckState)
  THEN
    _CheckStateLast:= _CheckState;
    _CheckTime     := F_GetTimeMsTick();
    (*-----------------------------------------------------------------------------------*)
    _CheckWorkFolder.sNetID   := '';   // local
    _CheckWorkFolder.sPathName:= _MainFolder;   // without trailing '/'
    _CheckWorkFolder.eCmd     := Tc2_Utilities.E_EnumCmdType.eEnumCmd_First;
    _CheckWorkFolder.tTimeout := Tc2_System.DEFAULT_ADS_TIMEOUT;
  END_IF

  (*-- ACTION ------------------------------------------------------------------------------------------------------------------*)

  (*-- TRANSITION --------------------------------------------------------------------------------------------------------------*)
  _CheckState:= E_TraceCheckStates.Scan;




(********************************************************************************************************************************)
(** check folder exists *********************************************************************************************************)
E_TraceCheckStates.Scan:
  (*-- ENTRY -------------------------------------------------------------------------------------------------------------------*)
  IF (_CheckStateLast <> _CheckState)
  THEN
    _CheckStateLast:= _CheckState;
    _CheckTime     := F_GetTimeMsTick();
    (*-----------------------------------------------------------------------------------*)
{warning disable C0139}
    _CheckWorkFolder( bExecute:= FALSE );
    _CheckWorkFolder.sNetID   ;   // hier nicht beschreiben
    _CheckWorkFolder.sPathName;   // hier nicht beschreiben
    _CheckWorkFolder.eCmd     ;   // hier nicht beschreiben
    _CheckWorkFolder.bExecute := TRUE;
    _CheckWorkFolder.tTimeout ;   // hier nicht beschreiben
{warning restore C0139}
  END_IF

  (*-- ACTION ------------------------------------------------------------------------------------------------------------------*)
  _CheckWorkFolder();

  (*-- TRANSITION --------------------------------------------------------------------------------------------------------------*)
  IF (_CheckWorkFolder.bBusy = FALSE)
  THEN
    _CheckWorkFolder.eCmd:= Tc2_Utilities.E_EnumCmdType.eEnumCmd_Next;
    (*-- Fehler -------------------------------------------------------------------------*)
    IF (_CheckWorkFolder.bError = TRUE)
    THEN
      //ErrorText:= 'target unreachable: ' + _WorkNetId.Value
      _Active    := FALSE;
      _CheckState:= E_TraceCheckStates.Wait;
    (*-- end of directory reached -------------------------------------------------------*)
    ELSIF (_CheckWorkFolder.bEOE = TRUE)
    THEN
      //ErrorText:= 'path not found: ' + _FilePath
      _Active    := FALSE;
      _CheckState:= E_TraceCheckStates.Wait;
    (*-- found as directory -------------------------------------------------------------*)
    ELSIF (_CheckWorkFolder.stFindFile.fileAttributes.bDirectory = TRUE)
    THEN
      //ErrorText:= '';
      _Active    := TRUE;
      _CheckState:= E_TraceCheckStates.Cancel;
    (*-- keep searching -----------------------------------------------------------------*)
    ELSE
      _CheckStateLast:= E_TraceCheckStates.Initialization;  // Re-entry
    END_IF

  END_IF




(********************************************************************************************************************************)
(********************************************************************************************************************************)
E_TraceCheckStates.Cancel:
  (*-- ENTRY -------------------------------------------------------------------------------------------------------------------*)
  IF (_CheckStateLast <> _CheckState)
  THEN
    _CheckStateLast:= _CheckState;
    _CheckTime     := F_GetTimeMsTick();
    (*-----------------------------------------------------------------------------------*)
{warning disable C0139}
    _CheckWorkFolder( bExecute:= FALSE );
    _CheckWorkFolder.sNetID;      // hier nicht beschreiben
    _CheckWorkFolder.sPathName;   // hier nicht beschreiben
    _CheckWorkFolder.eCmd     := Tc2_Utilities.E_EnumCmdType.eEnumCmd_Abort;
    _CheckWorkFolder.bExecute := TRUE;
    _CheckWorkFolder.tTimeout ;   // hier nicht beschreiben
{warning restore C0139}
  END_IF

  (*-- ACTION ------------------------------------------------------------------------------------------------------------------*)
  _CheckWorkFolder();

  (*-- TRANSITION --------------------------------------------------------------------------------------------------------------*)
  IF (_CheckWorkFolder.bBusy = FALSE)
  THEN
    (*-- error --------------------------------------------------------------------------*)
    IF (_CheckWorkFolder.bError = TRUE)
    THEN
      //ErrorText:= 'target unreachable'
      _Active    := FALSE;
      _CheckState:= E_TraceCheckStates.Wait;
    (*-- end of directory reached -------------------------------------------------------*)
    ELSIF (_CheckWorkFolder.bEOE = TRUE)
    THEN
      _CheckState:= E_TraceCheckStates.Wait;
    (*-- keep cancelling ----------------------------------------------------------------*)
    ELSE
      _CheckStateLast:= E_TraceCheckStates.Initialization;  // Re-entry
    END_IF
  END_IF




(********************************************************************************************************************************)
(********************************************************************************************************************************)
E_TraceCheckStates.Wait:
  (*-- ENTRY -------------------------------------------------------------------------------------------------------------------*)
  IF (_CheckStateLast <> _CheckState)
  THEN
    _CheckStateLast:= _CheckState;
    _CheckTime     := F_GetTimeMsTick();
    (*-----------------------------------------------------------------------------------*)
  END_IF

  (*-- ACTION ------------------------------------------------------------------------------------------------------------------*)

  (*-- TRANSITION --------------------------------------------------------------------------------------------------------------*)
  (*-- disabled -------------------------------------------------------------------------*)
  IF (_Enable = FALSE)
  THEN
    _CheckState:= E_TraceCheckStates.Disabled;
  (*-- wait time over -------------------------------------------------------------------*)
  ELSIF(F_GetTimeMsDiff(_CheckTime) >= T#1S)
  THEN
    _CheckState:= E_TraceCheckStates.HddCheck;
  END_IF




(********************************************************************************************************************************)
(** unknown *********************************************************************************************************************)
ELSE
  _CheckState:= E_TraceCheckStates.Initialization;
END_CASE




(********************************************************************************************************************************)
(** done ************************************************************************************************************************)
END_METHOD

// deletes all files and folders older than specified
METHOD PROTECTED M_RunDelete

(********************************************************************************************************************************)
VAR
  FolderDate            : TIMESTRUCT;
  (*----------------------------------------------------------------------------------------------------------------------------*)
  SystemTimeTD          : DATE_AND_TIME                    := DT#1979-01-09-23:59:59;
  FolderTimeTD          : DATE_AND_TIME                    := DT#1979-01-09-23:59:59;
  Diff_Seconds          : LINT                             := 0;
  (*----------------------------------------------------------------------------------------------------------------------------*)
  DestStart             : POINTER TO BYTE                  := 0;     // start position to concat
  DestEnd               : POINTER TO BYTE                  := 0;     // buffer/string end
  Result                : BOOL                             := FALSE;
END_VAR

(********************************************************************************************************************************)
(** initialization **************************************************************************************************************)
CASE(_DeleteState) OF
E_TraceDeleteStates.Initialization:
  (*-- ENTRY -------------------------------------------------------------------------------------------------------------------*)
    _DeleteStateLast:= _DeleteState;

  (*-- ACTION ------------------------------------------------------------------------------------------------------------------*)

  (*-- TRANSITION --------------------------------------------------------------------------------------------------------------*)
  _DeleteState:= E_TraceDeleteStates.WaitFolder;




(********************************************************************************************************************************)
(** wait working folder *********************************************************************************************************)
E_TraceDeleteStates.WaitFolder:
  (*-- ENTRY -------------------------------------------------------------------------------------------------------------------*)
  IF (_DeleteStateLast <> _DeleteState)
  THEN
    _DeleteStateLast:= _DeleteState;
    _DeleteTime     := F_GetTimeMsTick();
    (*-----------------------------------------------------------------------------------*)
  END_IF

  (*-- ACTION ------------------------------------------------------------------------------------------------------------------*)

  (*-- TRANSITION --------------------------------------------------------------------------------------------------------------*)
  (*-- working folder exists ------------------------------------------------------------*)
  IF (_Active = TRUE)
  THEN
    _DeleteState:= E_TraceDeleteStates.WaitDelay;
  END_IF




(********************************************************************************************************************************)
(** wait awhile *****************************************************************************************************************)
E_TraceDeleteStates.WaitDelay:
  (*-- ENTRY -------------------------------------------------------------------------------------------------------------------*)
  IF (_DeleteStateLast <> _DeleteState)
  THEN
    _DeleteStateLast:= _DeleteState;
    _DeleteTime     := F_GetTimeMsTick();
    (*-----------------------------------------------------------------------------------*)
  END_IF

  (*-- ACTION ------------------------------------------------------------------------------------------------------------------*)

  (*-- TRANSITION --------------------------------------------------------------------------------------------------------------*)
  (*-- working folder not existing ------------------------------------------------------*)
  IF (_Active = FALSE)
  THEN
    _DeleteState:= E_TraceDeleteStates.WaitFolder;
  (*-- delay time over ------------------------------------------------------------------*)
  ELSIF(F_GetTimeMsDiff(_DeleteTime) >= T#10S)
  THEN
    _DeleteState:= E_TraceDeleteStates.FolderStart;
  END_IF




(********************************************************************************************************************************)
(** prepare folder scan *********************************************************************************************************)
E_TraceDeleteStates.FolderStart:
  (*-- ENTRY -------------------------------------------------------------------------------------------------------------------*)
  IF (_DeleteStateLast <> _DeleteState)
  THEN
    _DeleteStateLast:= _DeleteState;
    _DeleteTime     := F_GetTimeMsTick();
    (*-- prepare folder scan ------------------------------------------------------------*)
    _ScanSubFolder.eCmd:= E_EnumCmdType.eEnumCmd_First;
  END_IF

  (*-- ACTION ------------------------------------------------------------------------------------------------------------------*)

  (*-- TRANSITION --------------------------------------------------------------------------------------------------------------*)
    _DeleteState:= E_TraceDeleteStates.FolderSeek;




(********************************************************************************************************************************)
(** find next (sub) folder ******************************************************************************************************)
E_TraceDeleteStates.FolderSeek:
  (*-- ENTRY -------------------------------------------------------------------------------------------------------------------*)
  IF (_DeleteStateLast <> _DeleteState)
  THEN
    _DeleteStateLast:= _DeleteState;
    _DeleteTime     := F_GetTimeMsTick();
    (*-----------------------------------------------------------------------------------*)
    _ScanSubFolder( bExecute:= FALSE );
    _ScanSubFolder.sNetID   := '';   // local
//  _ScanSubFolder.eCmd;   (* hier nicht beschreiben *)
    _ScanSubFolder.bExecute := TRUE;
    _ScanSubFolder.tTimeout := Tc2_System.DEFAULT_ADS_TIMEOUT;
    (*-----------------------------------------------------------------------------------*)
    DestStart:= ADR(_ScanSubFolder.sPathName);
    DestEnd  := ADR(_ScanSubFolder.sPathName) + SIZEOF(_ScanSubFolder.sPathName);
    DestStart:= F_StringCopy( DestStart:= DestStart,  DestEnd:= DestEnd,  Source:= ADR(_MainFolder)  );
    DestStart:= F_StringCopy( DestStart:= DestStart,  DestEnd:= DestEnd,  Source:= ADR('/*.*')  );
  END_IF

  (*-- ACTION ------------------------------------------------------------------------------------------------------------------*)
  _ScanSubFolder();

  (*-- TRANSITION --------------------------------------------------------------------------------------------------------------*)
  IF (_ScanSubFolder.bBusy = FALSE)
  THEN
    _ScanSubFolder.eCmd:= E_EnumCmdType.eEnumCmd_Next;
    (*-- error --------------------------------------------------------------------------*)
    IF    (_ScanSubFolder.bError = TRUE)
    THEN  (* unfortunately no difference between path noch found or destination not reachable *)
      _DeleteState:= E_TraceDeleteStates.WaitDelay;
    (*-- folder completely scanned ------------------------------------------------------*)
    ELSIF (_ScanSubFolder.bEOE = TRUE)
    THEN
      _DeleteState:= E_TraceDeleteStates.WaitDelay;
    (*-- found entry is no folder => continue -------------------------------------------*)
    ELSIF (_ScanSubFolder.stFindFile.fileAttributes.bDirectory = FALSE)
    THEN
      _DeleteStateLast:= E_TraceDeleteStates.Initialization;   // Re-entry
    (*-- folder name invalid => continue ------------------------------------------------*)
    ELSIF (    (_ScanSubFolder.stFindFile.sFileName = '.' )
            OR (_ScanSubFolder.stFindFile.sFileName = '..')  )
    THEN
      _DeleteStateLast:= E_TraceDeleteStates.Initialization;   // Re-entry
    (*-- folder valid => old enough to delete? ------------------------------------------*)
    ELSE
      (*-- parse folder name according to 'YYYY-MM-DD' --------------*)
      Result:= F_StringToTimeDate( AllowInvalidChars:= FALSE,  // invalid charachters will lead to parsing error
                                   DestStart        := ADR(_ScanSubFolder.stFindFile.sFileName),
                                   DestEnd          := ADR(_ScanSubFolder.stFindFile.sFileName) + SIZEOF(_ScanSubFolder.stFindFile.sFileName),
                                   Result     => FolderDate  );
      (*-- calc difference (in ms due to TIME limitation of 42d) ----*)
      SystemTimeTD:= SYSTEMTIME_TO_DT(System.fbSystemTime.TIMESTR);
      FolderTimeTD:= SYSTEMTIME_TO_DT(FolderDate);
      Diff_Seconds:= DT_TO_LINT(SystemTimeTD) - DT_TO_LINT(FolderTimeTD);
     (*-- folder name doesnt fit naming scheme YYYY-MM-DD -----------*)
      IF (Result = FALSE)
      THEN  // ignore ==> continue
        _DeleteStateLast:= E_TraceDeleteStates.Initialization;   // Re-entry
      (*-- folder from future ;-) -----------------------------------*)
      ELSIF (Diff_Seconds < 0)
      THEN  // ignore ==> continue
        _DeleteStateLast:= E_TraceDeleteStates.Initialization;   // Re-entry
      (*-- folder according parsed name too old ---------------------*)
      ELSIF (Diff_Seconds * 1_000 >= TIME_TO_LINT(SHELF_LIFE)  )  // TIME is internally already ms
      THEN  // => empty and delete
        _DeleteState:= E_TraceDeleteStates.FileStart;
      (*-- keep searching -------------------------------------------*)
      ELSE
        _DeleteStateLast:= E_TraceDeleteStates.Initialization;   // Re-entry
      END_IF
    END_IF
  END_IF




(********************************************************************************************************************************)
(** prepare file scan ***********************************************************************************************************)
E_TraceDeleteStates.FileStart:
  (*-- ENTRY -------------------------------------------------------------------------------------------------------------------*)
  IF (_DeleteStateLast <> _DeleteState)
  THEN
    _DeleteStateLast:= _DeleteState;
    _DeleteTime     := F_GetTimeMsTick();
    (*-----------------------------------------------------------------------------------*)
    _FileFind.eCmd:= E_EnumCmdType.eEnumCmd_First;
  END_IF

  (*-- ACTION ------------------------------------------------------------------------------------------------------------------*)

  (*-- TRANSITION --------------------------------------------------------------------------------------------------------------*)
  _DeleteState:= E_TraceDeleteStates.FileSeek;




(********************************************************************************************************************************)
(** find a file *****************************************************************************************************************)
E_TraceDeleteStates.FileSeek:
  (*-- ENTRY -------------------------------------------------------------------------------------------------------------------*)
  IF (_DeleteStateLast <> _DeleteState)
  THEN
    _DeleteStateLast:= _DeleteState;
    _DeleteTime     := F_GetTimeMsTick();
    (*-----------------------------------------------------------------------------------*)
    _FileFind( bExecute:= FALSE );
    _FileFind.sNetID   := '';   // local
//  _FileFind.eCmd;      (* hier nicht beschreiben *)
    _FileFind.bExecute := TRUE;
    _FileFind.tTimeout := Tc2_System.DEFAULT_ADS_TIMEOUT;
    (*-----------------------------------------------------------------------------------*)
    DestStart:= ADR(_FileFind.sPathName);
    DestEnd  := ADR(_FileFind.sPathName) + SIZEOF(_FileFind.sPathName);
    DestStart:= F_StringCopy( DestStart:= DestStart,  DestEnd:= DestEnd,  Source:= ADR(_MainFolder)  );
    DestStart:= F_StringCopy( DestStart:= DestStart,  DestEnd:= DestEnd,  Source:= ADR('/')  );
    DestStart:= F_StringCopy( DestStart:= DestStart,  DestEnd:= DestEnd,  Source:= ADR(_ScanSubFolder.stFindFile.sFileName)  );
    DestStart:= F_StringCopy( DestStart:= DestStart,  DestEnd:= DestEnd,  Source:= ADR('/*.*')  );
  END_IF

  (*-- ACTION ------------------------------------------------------------------------------------------------------------------*)
  _FileFind();

  (*-- TRANSITION --------------------------------------------------------------------------------------------------------------*)
  IF ( _FileFind.bBusy = FALSE )
  THEN
    _FileFind.eCmd:= E_EnumCmdType.eEnumCmd_Next;
    (*-- error --------------------------------------------------------------------------*)
    IF    (_FileFind.bError = TRUE)
    THEN
      _DeleteState:= E_TraceDeleteStates.WaitDelay;
    (*-- folder completely scanned ------------------------------------------------------*)
    ELSIF (_FileFind.bEOE = TRUE)
    THEN
      _DeleteState:= E_TraceDeleteStates.FolderDelete;
    (*-- file name invalid => continue --------------------------------------------------*)
    ELSIF (    (_FileFind.stFindFile.sFileName = '.' )
            OR (_FileFind.stFindFile.sFileName = '..')  )
    THEN
      _DeleteStateLast:= E_TraceDeleteStates.Initialization;   // Re-entry
    (*-- file found ==> delete ----------------------------------------------------------*)
    ELSE
      _DeleteState:= E_TraceDeleteStates.FileDelete;
    END_IF
  END_IF




(********************************************************************************************************************************)
(** delete this one file ********************************************************************************************************)
E_TraceDeleteStates.FileDelete:
  (*-- ENTRY -------------------------------------------------------------------------------------------------------------------*)
  IF (_DeleteStateLast <> _DeleteState)
  THEN
    _DeleteStateLast:= _DeleteState;
    _DeleteTime     := F_GetTimeMsTick();
    (*-----------------------------------------------------------------------------------*)
    _FileDelete( bExecute:= FALSE );
    _FileDelete.sNetId   := '';   // local
    _FileDelete.ePath    := E_OpenPath.PATH_GENERIC;  
    _FileDelete.bExecute := TRUE;
    _FileDelete.tTimeout := Tc2_System.DEFAULT_ADS_TIMEOUT;               
    (*-----------------------------------------------------------------------------------*)
    DestStart:= ADR(_FileDelete.sPathName);
    DestEnd  := ADR(_FileDelete.sPathName) + SIZEOF(_FileDelete.sPathName);
    DestStart:= F_StringCopy( DestStart:= DestStart,  DestEnd:= DestEnd,  Source:= ADR(_MainFolder)  );
    DestStart:= F_StringCopy( DestStart:= DestStart,  DestEnd:= DestEnd,  Source:= ADR('/')  );
    DestStart:= F_StringCopy( DestStart:= DestStart,  DestEnd:= DestEnd,  Source:= ADR(_ScanSubFolder.stFindFile.sFileName)  );
    DestStart:= F_StringCopy( DestStart:= DestStart,  DestEnd:= DestEnd,  Source:= ADR('/')  );
    DestStart:= F_StringCopy( DestStart:= DestStart,  DestEnd:= DestEnd,  Source:= ADR(_FileFind.stFindFile.sFileName)  );
  END_IF

  (*-- ACTION ------------------------------------------------------------------------------------------------------------------*)
  _FileDelete();

  (*-- TRANSITION --------------------------------------------------------------------------------------------------------------*)
  IF ( _FileDelete.bBusy = FALSE )
  THEN
    _DeleteState:= E_TraceDeleteStates.FileSeek;
  END_IF




(********************************************************************************************************************************)
(** delete that (now empty) folder **********************************************************************************************)
E_TraceDeleteStates.FolderDelete:
  (*-- ENTRY -------------------------------------------------------------------------------------------------------------------*)
  IF (_DeleteStateLast <> _DeleteState)
  THEN
    _DeleteStateLast:= _DeleteState;
    _DeleteTime     := F_GetTimeMsTick();
    (*-----------------------------------------------------------------------------------*)
    _FolderRemove( bExecute:= FALSE );
    _FolderRemove.sNetId   := '';   // local
    _FolderRemove.ePath    := E_OpenPath.PATH_GENERIC;
    _FolderRemove.bExecute := TRUE;
    _FolderRemove.tTimeout := Tc2_System.DEFAULT_ADS_TIMEOUT;
    (*-----------------------------------------------------------------------------------*)
    DestStart:= ADR(_FolderRemove.sPathName);
    DestEnd  := ADR(_FolderRemove.sPathName) + SIZEOF(_FolderRemove.sPathName);
    DestStart:= F_StringCopy( DestStart:= DestStart,  DestEnd:= DestEnd,  Source:= ADR(_MainFolder)  );
    DestStart:= F_StringCopy( DestStart:= DestStart,  DestEnd:= DestEnd,  Source:= ADR('/')  );
    DestStart:= F_StringCopy( DestStart:= DestStart,  DestEnd:= DestEnd,  Source:= ADR(_ScanSubFolder.stFindFile.sFileName)  );
    DestStart:= F_StringCopy( DestStart:= DestStart,  DestEnd:= DestEnd,  Source:= ADR('/')  );
  END_IF

  (*-- ACTION ------------------------------------------------------------------------------------------------------------------*)
  _FolderRemove();

  (*-- TRANSITION --------------------------------------------------------------------------------------------------------------*)
  IF ( _FolderRemove.bBusy = FALSE )
  THEN
    _DeleteState:= E_TraceDeleteStates.HddUsage;
    (*-- trace it ---------------------------------------------------*)
// example: '11-000-0000-00-0, old folder deleted,  folder = D:/Traces/1979-01-09/'
    _Text:= '';
    _Text:= CONCAT(_Text, F_AddDividerToSisString(SubsystemRegistry.SubsystemName) );
    _Text:= CONCAT(_Text, ',  old folder deleted');
    _Text:= CONCAT(_Text, DebugTextBlocks.FOLDER);
    _Text:= CONCAT(_Text, _FolderRemove.sPathName);
    Put( MsgType := E_DebugMsgType.INFO,
         Instance:= ADR(_Instance),
         Text    := ADR(_Text)  );
  END_IF




(********************************************************************************************************************************)
(** read current hdd usage ******************************************************************************************************)
E_TraceDeleteStates.HddUsage:
  (*-- ENTRY -------------------------------------------------------------------------------------------------------------------*)
  IF (_DeleteStateLast <> _DeleteState)
  THEN
    _DeleteStateLast:= _DeleteState;
    _DeleteTime     := F_GetTimeMsTick();
    (*-----------------------------------------------------------------------------------*)
    _HddUsage.Start( Drive:= _MainFolder );  // use drive letter from main folder
  END_IF

  (*-- ACTION ------------------------------------------------------------------------------------------------------------------*)

  (*-- TRANSITION --------------------------------------------------------------------------------------------------------------*)
  IF (_HddUsage.Busy = FALSE)
  THEN
    _HddUsageCount:= _HddUsageCount + 1;
    _HddStateLast := E_TraceHddUsageStates.Initialization;  // force re-entry and write message
    (*-------------------------------------------*)
    _DeleteState:= E_TraceDeleteStates.FolderSeek;
  END_IF




(********************************************************************************************************************************)
(** unknown *********************************************************************************************************************)
ELSE
  _DeleteState:= E_TraceDeleteStates.Initialization;
END_CASE




(********************************************************************************************************************************)
(** done ************************************************************************************************************************)
END_METHOD

// creates hdd usage debug messages
METHOD PROTECTED M_RunHddUsage

(********************************************************************************************************************************)
VAR
END_VAR

(********************************************************************************************************************************)
(** diagnosis *******************************************************************************************************************)
{warning disable C0139}
_HddUsage.BytesTotal;
_HddUsage.BytesUsed;    _HddUsage.PercentageUsed;
_HddUsage.BytesFree;    _HddUsage.PercentageFree;
{warning restore C0139}




(********************************************************************************************************************************)
(** initialisation **************************************************************************************************************)
CASE (_HddState) OF
E_TraceHddUsageStates.Initialization:
  (*-- ENTRY -------------------------------------------------------------------------------------------------------------------*)
    _HddStateLast:= _HddState;
    _HddTooFull  := FALSE;

  (*-- ACTION ------------------------------------------------------------------------------------------------------------------*)

  (*-- TRANSITION --------------------------------------------------------------------------------------------------------------*)
    // takes place in state E_TraceCheckStates.HddUsage of M_RunCheck()




(********************************************************************************************************************************)
(** unknown *********************************************************************************************************************)
E_TraceHddUsageStates.Unknown:
  (*-- ENTRY -------------------------------------------------------------------------------------------------------------------*)
  IF (_HddStateLast <> _HddState)
  THEN
    _HddStateLast:= _HddState;
    _HddTooFull  := FALSE;
    (*-----------------------------------------------------------------------------------*)
    // example: '11-000-0000-00-0, unable to retrieve hdd usage,  drive = D:/'
    _Text:= '';
    _Text:= CONCAT(_Text, F_AddDividerToSisString(SubsystemRegistry.SubsystemName) );
    _Text:= CONCAT(_Text, ',  unable to retrieve hdd usage');
    _Text:= CONCAT(_Text, DebugTextBlocks.DRIVE);
    _Text:= CONCAT(_Text, _HddUsage.Drive);
    IF (_HddFullMissed <> 0)
    THEN
      _Text:= CONCAT(_Text, DebugTextBlocks.MISSED);  _Text:= CONCAT(_Text, ULINT_TO_STRING(_HddFullMissed)   );
    END_IF
    Put( MsgType := E_DebugMsgType.ERROR,
         Instance:= ADR(_Instance),
         Text    := ADR(_Text)  );
    (*-----------------------------------------------------------------------------------*)
    _HddFullMissed:= 0;
  END_IF

  (*-- ACTION ------------------------------------------------------------------------------------------------------------------*)

  (*-- TRANSITION --------------------------------------------------------------------------------------------------------------*)
    // takes place in state E_TraceCheckStates.HddUsage of M_RunCheck()




(********************************************************************************************************************************)
(** enough space free ***********************************************************************************************************)
E_TraceHddUsageStates.EnoughFree:
  (*-- ENTRY -------------------------------------------------------------------------------------------------------------------*)
  IF (_HddStateLast <> _HddState)
  THEN
    _HddStateLast:= _HddState;
    _HddTooFull  := FALSE;
    (*-----------------------------------------------------------------------------------*)
    // example: '11-000-0000-00-0, hdd usage information,  drive = D:/:,  total = 320GB,  free = 98GB,  usage = 65%'
    _Text:= '';
    _Text:= CONCAT(_Text, F_AddDividerToSisString(SubsystemRegistry.SubsystemName) );
    _Text:= CONCAT(_Text, ',  hdd usage information');
    _Text:= CONCAT(_Text, DebugTextBlocks.DRIVE);  _Text:= CONCAT(_Text, _HddUsage.Drive);
    _Text:= CONCAT(_Text, DebugTextBlocks.TOTAL);  _Text:= CONCAT(_Text, F_DiskSpaceToString(_HddUsage.BytesTotal)  );
    _Text:= CONCAT(_Text, DebugTextBlocks.FREE);   _Text:= CONCAT(_Text, F_DiskSpaceToString(_HddUsage.BytesFree)   );
    _Text:= CONCAT(_Text, DebugTextBlocks.USED);   _Text:= CONCAT(_Text, F_DiskSpaceToString(_HddUsage.BytesUsed)   );
    _Text:= CONCAT(_Text, DebugTextBlocks.USAGE);  _Text:= CONCAT(_Text, BYTE_TO_STRING(_HddUsage.PercentageUsed)   );  _Text:= CONCAT(_Text, '%');
    IF (_HddFullMissed <> 0)
    THEN
      _Text:= CONCAT(_Text, DebugTextBlocks.MISSED);  _Text:= CONCAT(_Text, ULINT_TO_STRING(_HddFullMissed)   );
    END_IF
    Put( MsgType := E_DebugMsgType.INFO,
         Instance:= ADR(_Instance),
         Text    := ADR(_Text)  );
    (*-----------------------------------------------------------------------------------*)
    _HddFullMissed:= 0;
  END_IF

  (*-- ACTION ------------------------------------------------------------------------------------------------------------------*)

  (*-- TRANSITION --------------------------------------------------------------------------------------------------------------*)
    // takes place in state E_TraceCheckStates.HddUsage of M_RunCheck()




(********************************************************************************************************************************)
(** warning level ***************************************************************************************************************)
E_TraceHddUsageStates.WarningLevel:
  (*-- ENTRY -------------------------------------------------------------------------------------------------------------------*)
  IF (_HddStateLast <> _HddState)
  THEN
    _HddStateLast:= _HddState;
    _HddTooFull  := FALSE;
    (*-----------------------------------------------------------------------------------*)
    // example: '11-000-0000-00-0, hdd usage information,  drive = D:/:,  total = 320GB,  free = 98GB,  usage = 65%,  missed messages = 1234'
    _Text:= '';
    _Text:= CONCAT(_Text, F_AddDividerToSisString(SubsystemRegistry.SubsystemName) );
    _Text:= CONCAT(_Text, ',  hdd usage information');
    _Text:= CONCAT(_Text, DebugTextBlocks.DRIVE);  _Text:= CONCAT(_Text, _HddUsage.Drive);
    _Text:= CONCAT(_Text, DebugTextBlocks.TOTAL);  _Text:= CONCAT(_Text, F_DiskSpaceToString(_HddUsage.BytesTotal)  );
    _Text:= CONCAT(_Text, DebugTextBlocks.FREE);   _Text:= CONCAT(_Text, F_DiskSpaceToString(_HddUsage.BytesFree)   );
    _Text:= CONCAT(_Text, DebugTextBlocks.USED);   _Text:= CONCAT(_Text, F_DiskSpaceToString(_HddUsage.BytesUsed)   );
    _Text:= CONCAT(_Text, DebugTextBlocks.USAGE);  _Text:= CONCAT(_Text, BYTE_TO_STRING(_HddUsage.PercentageUsed)   );  _Text:= CONCAT(_Text, '%');
    IF (_HddFullMissed <> 0)
    THEN
      _Text:= CONCAT(_Text, DebugTextBlocks.MISSED);  _Text:= CONCAT(_Text, ULINT_TO_STRING(_HddFullMissed)   );
    END_IF
    Put( MsgType := E_DebugMsgType.WARNING,
         Instance:= ADR(_Instance),
         Text    := ADR(_Text)  );
    (*-----------------------------------------------------------------------------------*)
    _HddFullMissed:= 0;
  END_IF

  (*-- ACTION ------------------------------------------------------------------------------------------------------------------*)

  (*-- TRANSITION --------------------------------------------------------------------------------------------------------------*)
    // takes place in state E_TraceCheckStates.HddUsage of M_RunCheck()




(********************************************************************************************************************************)
(** error level *****************************************************************************************************************)
E_TraceHddUsageStates.ErrorLevel:
  (*-- ENTRY -------------------------------------------------------------------------------------------------------------------*)
  IF (_HddStateLast <> _HddState)
  THEN
    _HddStateLast:= _HddState;
    (*-----------------------------------------------------------------------------------*)
    // example: '11-000-0000-00-0, hdd usage information,  drive = D:/:,  total = 320GB,  free = 98GB,  usage = 65%'
    _Text:= '';
    _Text:= CONCAT(_Text, F_AddDividerToSisString(SubsystemRegistry.SubsystemName) );
    _Text:= CONCAT(_Text, ',  hdd usage information');
    _Text:= CONCAT(_Text, DebugTextBlocks.DRIVE);  _Text:= CONCAT(_Text, _HddUsage.Drive);
    _Text:= CONCAT(_Text, DebugTextBlocks.TOTAL);  _Text:= CONCAT(_Text, F_DiskSpaceToString(_HddUsage.BytesTotal)  );
    _Text:= CONCAT(_Text, DebugTextBlocks.FREE);   _Text:= CONCAT(_Text, F_DiskSpaceToString(_HddUsage.BytesFree)   );
    _Text:= CONCAT(_Text, DebugTextBlocks.USED);   _Text:= CONCAT(_Text, F_DiskSpaceToString(_HddUsage.BytesUsed)   );
    _Text:= CONCAT(_Text, DebugTextBlocks.USAGE);  _Text:= CONCAT(_Text, BYTE_TO_STRING(_HddUsage.PercentageUsed)   );  _Text:= CONCAT(_Text, '%');
    Put( MsgType := E_DebugMsgType.ERROR,
         Instance:= ADR(_Instance),
         Text    := ADR(_Text)  );
    (*-----------------------------------------------------------------------------------*)
    _HddTooFull   := TRUE; // after this Put() just above
    _HddFullMissed:= 0;
  END_IF

  (*-- ACTION ------------------------------------------------------------------------------------------------------------------*)

  (*-- TRANSITION --------------------------------------------------------------------------------------------------------------*)
    // takes place in state E_TraceCheckStates.HddUsage of M_RunCheck()




(********************************************************************************************************************************)
(** unknown *********************************************************************************************************************)
ELSE
  _HddState:= E_TraceHddUsageStates.Initialization;
END_CASE




(********************************************************************************************************************************)
(** done ************************************************************************************************************************)
END_METHOD

// writes traces into file
METHOD PROTECTED M_RunWrite

(********************************************************************************************************************************)
VAR
  DestStart             : POINTER TO BYTE                  := 0;     // start position to concat
  DestEnd               : POINTER TO BYTE                  := 0;     // buffer/string end
END_VAR

(********************************************************************************************************************************)
(** initialization **************************************************************************************************************)
CASE(_WriteState) OF
E_TraceWriteStates.Initialization:
  (*-- ENTRY -------------------------------------------------------------------------------------------------------------------*)
    _WriteStateLast:= _WriteState;

  (*-- ACTION ------------------------------------------------------------------------------------------------------------------*)

  (*-- TRANSITION --------------------------------------------------------------------------------------------------------------*)
  _WriteState:= E_TraceWriteStates.WaitFolder;




(********************************************************************************************************************************)
(** error - wait to disable *****************************************************************************************************)
E_TraceWriteStates.Error:
  (*-- ENTRY -------------------------------------------------------------------------------------------------------------------*)
  IF (_WriteStateLast <> _WriteState)
  THEN
    _WriteStateLast:= _WriteState;
    _WriteTime     := F_GetTimeMsTick();
    (*-----------------------------------------------------------------------------------*)
  END_IF

  (*-- ACTION ------------------------------------------------------------------------------------------------------------------*)

  (*-- TRANSITION --------------------------------------------------------------------------------------------------------------*)
  (*-- working folder dissapeared -------------------------------------------------------*)
  IF (_Active = FALSE)
  THEN
    _WriteState:= E_TraceWriteStates.WaitFolder;
  END_IF




(********************************************************************************************************************************)
(** wait working folder *********************************************************************************************************)
E_TraceWriteStates.WaitFolder:
  (*-- ENTRY -------------------------------------------------------------------------------------------------------------------*)
  IF (_WriteStateLast <> _WriteState)
  THEN
    _WriteStateLast:= _WriteState;
    _WriteTime     := F_GetTimeMsTick();
    (*-----------------------------------------------------------------------------------*)
  END_IF

  (*-- ACTION ------------------------------------------------------------------------------------------------------------------*)

  (*-- TRANSITION --------------------------------------------------------------------------------------------------------------*)
  (*-- working folder exists ------------------------------------------------------------*)
  IF (_Active = TRUE)
  THEN
    _WriteState:= E_TraceWriteStates.StartWork;
  END_IF




(********************************************************************************************************************************)
(** build working folder name with date *****************************************************************************************)
E_TraceWriteStates.StartWork:
  (*-- ENTRY -------------------------------------------------------------------------------------------------------------------*)
  IF (_WriteStateLast <> _WriteState)
  THEN
    _WriteStateLast:= _WriteState;
    _WriteTime     := F_GetTimeMsTick();
    (*-- save current working date ------------------------------------------------------*)
    _WriteDate:= System.fbSystemTime.TIMESTR;
    (*-- build folder name --------------------------------------------------------------*)
    DestStart:= ADR(_WritePath);
    DestEnd  := ADR(_WritePath) + SIZEOF(_WritePath);
    DestStart:= F_StringCopy          ( DestStart:= DestStart,  DestEnd:= DestEnd,  Source    := ADR(_MainFolder)  );
    DestStart:= F_StringCopy          ( DestStart:= DestStart,  DestEnd:= DestEnd,  Source    := ADR('/')  );
    DestStart:= F_StringFromDatestruct( DestStart:= DestStart,  DestEnd:= DestEnd,  DateStruct:= _WriteDate );
    DestStart:= F_StringCopy          ( DestStart:= DestStart,  DestEnd:= DestEnd,  Source    := ADR('/')  );
  END_IF

  (*-- ACTION ------------------------------------------------------------------------------------------------------------------*)

  (*-- TRANSITION --------------------------------------------------------------------------------------------------------------*)
  _WriteState:= E_TraceWriteStates.CreateDir;




(********************************************************************************************************************************)
(** create daily working folder *************************************************************************************************)
E_TraceWriteStates.CreateDir:
  (*-- ENTRY -------------------------------------------------------------------------------------------------------------------*)
  IF (_WriteStateLast <> _WriteState)
  THEN
    _WriteStateLast:= _WriteState;
    _WriteTime     := F_GetTimeMsTick();
    (*-----------------------------------------------------------------------------------*)
    _CreateDir( bExecute:= FALSE );         
    _CreateDir.sNetId   := '';  // local
    _CreateDir.sPathName:= _WritePath;
    _CreateDir.ePath    := E_OpenPath.PATH_GENERIC;
    _CreateDir.bExecute := TRUE;         
    _CreateDir.tTimeout := Tc2_System.DEFAULT_ADS_TIMEOUT;
  END_IF

  (*-- ACTION ------------------------------------------------------------------------------------------------------------------*)
  _CreateDir();

